TYPE ST_MotionData EXTENDS Tc2_MC2.NCTOPLC_AXIS_REF : 
STRUCT
	record_time : ULINT; 
END_STRUCT
END_TYPE

(* stored: Version 1.1.0.1, ProductVersion 3.1.4024.15
   DUT ST_MotionData: Id {957f2ee4-797d-497d-adf5-2f9c4f103a47} *)
